# EPICS autosave request: support/ebrick/2-2-3/iocBoot/iocebrick/autosave/ccdFunc_settings.req
$(P)$(E)$(F)$(T)
$(P)$(E)$(F)$(T):units
$(P)$(E)$(F)$(T):name
